// TIA Portal V19 export
VAR_GLOBAL   // PLC tag table "U2Em3_Inputs"
   hookClawCylinderHomePositionDetectionU2Em3_2 AT %I173.5 : Bool;   // U2Em3_ Hook claw cylinder 2 in-situ detection / Em100_钩爪气缸2原位检测
   hookClawCylinderWorkPositionDetectionU2Em3_2 AT %I173.4 : Bool;   // U2Em3_Hook claw cylinder 2 working position detection / Em100_钩爪气缸2工作位检测
   hookClawCylinderWorkPositionDetectionU2Em3_1 AT %I173.2 : Bool;   // U2Em3_Hook claw cylinder 1 working position detection / Em100_钩爪气缸1工作位检测
   slideCylinderWorkPositionDetectionU2Em3_1 AT %I172.1 : Bool;   // U2Em3_ Sliding table cylinder working position detection 1 / Em100_滑台气缸工作位检测1
   "null(21)" AT %I172.7 : Bool;   // 备用
   "null(22)" AT %I173.0 : Bool;   // 备用
   pressureGaugeSetValueDetectionU2Em3_1_2 AT %I170.3 : Bool;   // U2Em3_ Pressure gauge 1 set value detection 2 / Em100_压力表1设定值检测2
   slideCylinderMedianPositionDetectionU2Em3_1 AT %I172.3 : Bool;   // U2Em3_Middle position detection of slide cylinder 1 / Em100_滑台气缸中位检测1
   pressureGaugeSetValueDetectionU2Em3_1_1 AT %I170.2 : Bool;   // U2Em3_ Pressure gauge 1 set value detection 1 / Em100_压力表1设定值检测1
   motorConstraintOrgU2Em3_2 AT %I171.5 : Bool;   // U2Em3_Constrained Motor 2 Origin / Em100_拘束电机2原点
   hookClawCylinderHomePositionDetectionU2Em3_1 AT %I173.3 : Bool;   // U2Em3_ Hook claw cylinder 1 in-situ detection / Em100_钩爪气缸1原位检测
   slideCylinderWorkPositionDetectionU2Em3_2 AT %I172.4 : Bool;   // U2Em3_ Sliding table cylinder working position detection 2 / Em100_滑台气缸工作位检测2
   "null(28)" AT %I170.6 : Bool;   // 备用
   motorConstraintPotU2Em3_2 AT %I171.3 : Bool;   // U2Em3_ Restraint motor 2 positive limit / Em100_拘束电机2正限
   motorConstraintPotU2Em3_1 AT %I171.0 : Bool;   // U2Em3_ Restraint motor 1 positive limit / Em100_拘束电机1正限
   slideCylinderHomePositionDetectionU2Em3_1 AT %I172.2 : Bool;   // U2Em3_skid table cylinder in-situ detection 1 / Em100_滑台气缸原位检测1
   motorConstraintOrgU2Em3_1 AT %I171.2 : Bool;   // U2Em3_Constrained Motor 1 Origin / Em100_拘束电机1原点
   "null(23)" AT %I173.1 : Bool;   // 备用
   motorConstraintNotU2Em3_1 AT %I171.1 : Bool;   // U2Em3_ Restraint motor 1 negative limit / Em100_拘束电机1负限
   pressureGaugeSetValueDetectionU2Em3_2_2 AT %I170.5 : Bool;   // U2Em3_ Pressure gauge 2 set value detection 2 / Em100_压力表2设定值检测2
   pressureGaugeSetValueDetectionU2Em3_2_1 AT %I170.4 : Bool;   // U2Em3_ Pressure gauge 2 set value detection 1 / Em100_压力表2设定值检测1
   motorConstraintNotU2Em3_2 AT %I171.4 : Bool;   // U2Em3_ Restraint motor 2 negative limit / Em100_拘束电机2负限
   slideCylinderHomePositionDetectionU2Em3_2 AT %I172.5 : Bool;   // U2Em3_skid table cylinder in-situ detection 2 / Em100_滑台气缸原位检测2
   "null(20)" AT %I172.0 : Bool;   // 备用
   slideCylinderMedianPositionDetectionU2Em3_2 AT %I172.6 : Bool;   // U2Em3_Middle position detection of slide cylinder 2 / Em100_滑台气缸中位检测2
   "null(29)" AT %I170.7 : Bool;   // spare / 备用
   "null(25)" AT %I173.7 : Bool;   // spare / 备用
   "null(24)" AT %I173.6 : Bool;   // spare / 备用
END_VAR
